// TIA Portal V15.1 export
// export: Created 2024-06-21T08:40:36.5770637Z, ExportSetting WithDefaults, DisplayName Totally Integrated Automation Portal, DisplayVersion V15.1 Update 5, DisplayName TIA Portal Openness, DisplayVersion V15.1 Update 5, DisplayName SINAMICS Startdrive Advanced, DisplayVersion V15.1, DisplayName G130, G150, S120, S150, SINAMICS MV, S210, DisplayVersion V15.1, DisplayName G110M, G120, G120C, G120D, G120P, DisplayVersion V15.1, DisplayName STEP 7 Professional, DisplayVersion V15.1 Update 5, DisplayName STEP 7 Safety, DisplayVersion V15.1, DisplayName WinCC Professional, DisplayVersion V15.1 Update 5, DisplayName SIMATIC Visualization Architect, DisplayVersion V15.1
ORGANIZATION_BLOCK "CYC_INT2"   // OB32, FBD, CyclicInterrupt
TITLE = CYC_INT2
{ S7_Optimized_Access := 'TRUE' }
AUTHOR : VCC
VERSION : 0.0.0.0
// =============================================================================Cyclic Interrupt
// =============================================================================
// stored: AutoNumber false, IsIECCheckEnabled false, SetENOAutomatically False
   VAR_INPUT
      Initial_Call : Bool;   // Initial call of this OB
      Event_Count : Int;   // Events discarded
   END_VAR
BEGIN
END_ORGANIZATION_BLOCK
